(* IEC 61131-3 sources: OpenPLC/build, 2 files *)

(* ---- plc.st ---- *)
TYPE
  LOGLEVEL : (CRITICAL, WARNING, INFO, DEBUG) := INFO;
END_TYPE

FUNCTION_BLOCK LOGGER
  VAR_INPUT
    TRIG : BOOL;
    MSG : STRING;
    LEVEL : LOGLEVEL := INFO;
  END_VAR
  VAR
    TRIG0 : BOOL;
  END_VAR

  IF TRIG AND NOT TRIG0 THEN
  {{
   LogMessage(GetFbVar(LEVEL),(char*)GetFbVar(MSG, .body),GetFbVar(MSG, .len));
  }}
  END_IF;
  TRIG0:=TRIG;
END_FUNCTION_BLOCK

FUNCTION_BLOCK python_eval
  VAR_INPUT
    TRIG : BOOL;
    CODE : STRING;
  END_VAR
  VAR_OUTPUT
    ACK : BOOL;
    RESULT : STRING;
  END_VAR
  VAR
    STATE : DWORD;
    BUFFER : STRING;
    PREBUFFER : STRING;
    TRIGM1 : BOOL;
    TRIGGED : BOOL;
  END_VAR

  {extern void __PythonEvalFB(int, PYTHON_EVAL*);__PythonEvalFB(0, data__);}
END_FUNCTION_BLOCK

FUNCTION_BLOCK python_poll
  VAR_INPUT
    TRIG : BOOL;
    CODE : STRING;
  END_VAR
  VAR_OUTPUT
    ACK : BOOL;
    RESULT : STRING;
  END_VAR
  VAR
    STATE : DWORD;
    BUFFER : STRING;
    PREBUFFER : STRING;
    TRIGM1 : BOOL;
    TRIGGED : BOOL;
  END_VAR

  {extern void __PythonEvalFB(int, PYTHON_EVAL*);__PythonEvalFB(1,(PYTHON_EVAL*)(void*)data__);}
END_FUNCTION_BLOCK

FUNCTION_BLOCK python_gear
  VAR_INPUT
    N : UINT;
    TRIG : BOOL;
    CODE : STRING;
  END_VAR
  VAR_OUTPUT
    ACK : BOOL;
    RESULT : STRING;
  END_VAR
  VAR
    py_eval : python_eval;
    COUNTER : UINT;
    _TMP_ADD10_OUT : UINT;
    _TMP_EQ13_OUT : BOOL;
    _TMP_SEL15_OUT : UINT;
    _TMP_AND7_OUT : BOOL;
  END_VAR

  _TMP_ADD10_OUT := ADD(COUNTER, 1);
  _TMP_EQ13_OUT := EQ(N, _TMP_ADD10_OUT);
  _TMP_SEL15_OUT := SEL(_TMP_EQ13_OUT, _TMP_ADD10_OUT, 0);
  COUNTER := _TMP_SEL15_OUT;
  _TMP_AND7_OUT := AND(_TMP_EQ13_OUT, TRIG);
  py_eval(TRIG := _TMP_AND7_OUT, CODE := CODE);
  ACK := py_eval.ACK;
  RESULT := py_eval.RESULT;
END_FUNCTION_BLOCK

PROGRAM prueba
  VAR
    sensor_hall : BOOL := 0;
    led : BOOL := 1;
    led_rojo : BOOL := 0;
    rele : BOOL := 0;
  END_VAR
  VAR
    subir_pist : TP;
    counter : CTU;
    delay : TON;
    bajar_pist : TP;
    _TMP_NOT10_OUT : BOOL;
    R_TRIG1 : R_TRIG;
    _TMP_NOT16_OUT : BOOL;
  END_VAR

  _TMP_NOT10_OUT := NOT(sensor_hall);
  R_TRIG1(CLK := _TMP_NOT10_OUT);
  delay(IN := counter.Q, PT := T#12000ms);
  counter(CU := R_TRIG1.Q, R := delay.Q, PV := 5);
  subir_pist(IN := counter.Q, PT := T#2000ms);
  bajar_pist(IN := delay.Q, PT := T#2000ms);
  rele := bajar_pist.Q OR subir_pist.Q;
  led_rojo := counter.Q;
  _TMP_NOT16_OUT := NOT(counter.Q);
  led := _TMP_NOT16_OUT OR _TMP_NOT16_OUT;
END_PROGRAM

CONFIGURATION Config0

  RESOURCE Res0 ON PLC
    TASK task0(INTERVAL := T#20ms,PRIORITY := 0);
    PROGRAM instance0 WITH task0 : prueba;
  END_RESOURCE
END_CONFIGURATION

(* ---- generated_plc.st ---- *)
PROGRAM prueba
  VAR
    sensor_hall AT %IX0.0 : BOOL := 0;
    led AT %QX0.0 : BOOL := 1;
    led_rojo AT %QX0.2 : BOOL := 0;
    rele AT %QX0.1 : BOOL := 0;
  END_VAR
  VAR
    subir_pist : TP;
    counter : CTU;
    delay : TON;
    bajar_pist : TP;
    _TMP_NOT10_OUT : BOOL;
    R_TRIG1 : R_TRIG;
    _TMP_NOT16_OUT : BOOL;
  END_VAR

  _TMP_NOT10_OUT := NOT(sensor_hall);
  R_TRIG1(CLK := _TMP_NOT10_OUT);
  delay(IN := counter.Q, PT := T#12000ms);
  counter(CU := R_TRIG1.Q, R := delay.Q, PV := 5);
  subir_pist(IN := counter.Q, PT := T#2000ms);
  bajar_pist(IN := delay.Q, PT := T#2000ms);
  rele := bajar_pist.Q OR subir_pist.Q;
  led_rojo := counter.Q;
  _TMP_NOT16_OUT := NOT(counter.Q);
  led := _TMP_NOT16_OUT OR _TMP_NOT16_OUT;
END_PROGRAM

CONFIGURATION Config0

  RESOURCE Res0 ON PLC
    TASK task0(INTERVAL := T#20ms,PRIORITY := 0);
    PROGRAM instance0 WITH task0 : prueba;
  END_RESOURCE
END_CONFIGURATION
